{attribute addProperty BoxType "EKM1101-0000-0016"}
{attribute addProperty Id "ErrorBIT10.1251UnderrangeBIT10.1252OverrangeBIT10.1253DiagBIT10.1254Sensor_OvrBIT10.1255OverrunBIT10.1256TxPDO_StateBIT10.12515"}
{attribute addProperty CRC "1725206741"}
{attribute addProperty SizeInBites "16"}
{attribute addProperty SizeInBytes "2"}
TYPE Status_66D490D5 :
STRUCT
	{attribute addProperty Name "Error"}
	Error : BOOL;
	{attribute addProperty Name "Underrange"}
	Underrange : BOOL;
	{attribute addProperty Name "Overrange"}
	Overrange : BOOL;
	{attribute addProperty Name "Diag"}
	Diag : BOOL;
	{attribute addProperty Name "Sensor_Ovr"}
	Sensor_Ovr : BOOL;
	{attribute addProperty Name "Overrun"}
	Overrun : BOOL;
	{attribute 'hide'}
	reserve_1 : BYTE;
	{attribute addProperty Name "TxPDO_State"}
	TxPDO_State : BOOL;
	{attribute 'hide'}
	reserve_2 : BOOL;
END_STRUCT
END_TYPE

(* stored: Version 1.2.0.0, ProductVersion 3.1.4024.9
   DUT Status_66D490D5: Id {d3b0e01d-a232-4b2f-a5f7-c9169edc1b88} *)
